// LS Electric XG5000 project: Reset_이중코일문제
// PLC NewPLC
// module base 0 slot 0: 입출력 모듈:XBC-DR20S (DC 24V 입력 12점, 릴레이 출력 8점)

PROGRAM NewProgram (task: 스캔 프로그램)

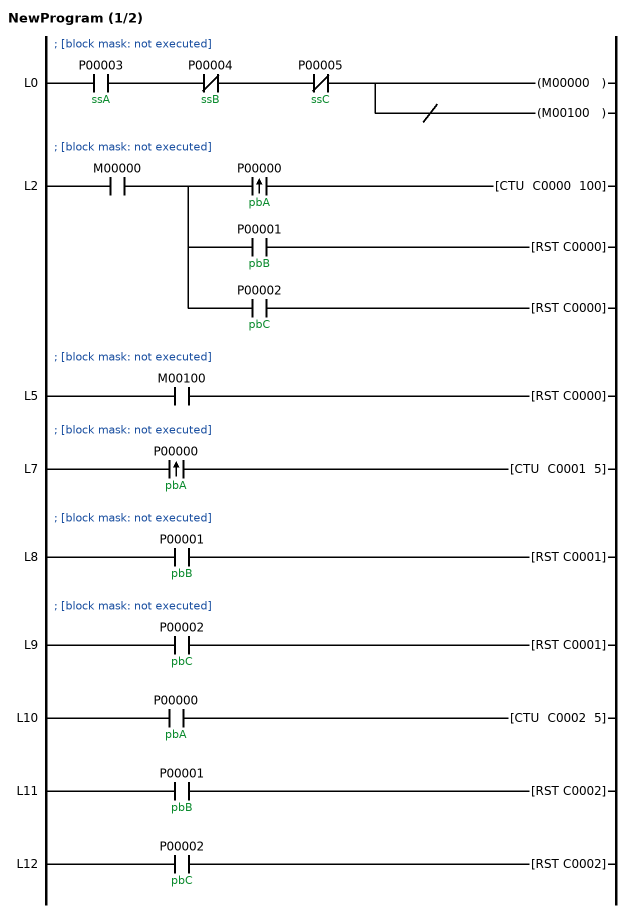
; L0 (block mask: not executed)
LOAD      P00003	// ssA
AND NOT   P00004	// ssB
AND NOT   P00005	// ssC
OUT       M00000
NOT
OUT       M00100
; L2 (block mask: not executed)
LOAD      M00000
MPUSH
ANDP      P00000	// pbA
CTU       C0000 100
MLOAD
AND       P00001	// pbB
RST       C0000
MPOP
AND       P00002	// pbC
RST       C0000
; L5 (block mask: not executed)
LOAD      M00100
RST       C0000
; L7 (block mask: not executed)
LOADP     P00000	// pbA
CTU       C0001 5
; L8 (block mask: not executed)
LOAD      P00001	// pbB
RST       C0001
; L9 (block mask: not executed)
LOAD      P00002	// pbC
RST       C0001
; L10
LOAD      P00000	// pbA
CTU       C0002 5
; L11
LOAD      P00001	// pbB
RST       C0002
; L12
LOAD      P00002	// pbC
RST       C0002

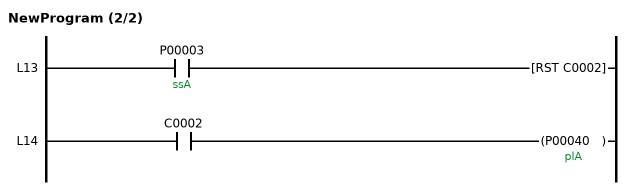
; L13
LOAD      P00003	// ssA
RST       C0002
; L14
LOAD      C0002
OUT       P00040	// plA

VARIABLES AND COMMENTS (devices not used above)
P00041	BIT	plB
P00042	BIT	plC
P00043	BIT	plD
P00044	BIT	plE